// TIA Portal project "Esteira Properzi" (V15)

(* hardware
DEVICE "S7-1200 station_1"  S7-1200 Station
   slot 0: "Rack_0"  S7-1200 Rack  Rack  V1.0
   slot 1: "PLC_1"  CPU 1214C DC/DC/DC  6ES7 214-1AG40-0XB0  V4.2
*)

// ===== PLC "PLC_1"  CPU 1214C DC/DC/DC =====

VAR_GLOBAL   // PLC tag table "Default tag table"
   "Sensor Inicio Esteira" AT %I0.0 : Bool;
   "Sensor Meio Esteira" AT %I0.1 : Bool;
   "Sensor Fim Esteira" AT %I0.2 : Bool;
   "Sensor Nivel Alto Fusao" AT %I0.3 : Bool;
   "Sensor Nivel Medio Fusao" AT %I0.4 : Bool;
   "Sensor Nivel Baixo Fusao" AT %I0.5 : Bool;
   "Emergencia" AT %I0.6 : Bool;
   "Aut \ Man" AT %I0.7 : Bool;
   "Liga" AT %I1.0 : Bool;
   "Desliga" AT %I1.1 : Bool;
   "Motor" AT %Q0.0 : Bool;
   "Sinaleiro Verde" AT %Q0.1 : Bool;
   "Sinaleiro Vermelho" AT %Q0.2 : Bool;
   "Sonorizador" AT %Q0.3 : Bool;
   "Aux Sensor Inicio Esteira" AT %M2.0 : Bool;
   "Aux Sensor Meio Esteira" AT %M2.1 : Bool;
   "Aux Sensor Fim Esteira" AT %M2.2 : Bool;
   "Aux Sensor Nivel Alto Fusao" AT %M2.3 : Bool;
   "Aux Sensor Nivel Medio Fusao" AT %M2.4 : Bool;
   "Aux Sensor Nivel Baixo Fusao" AT %M2.5 : Bool;
   "System_Byte" AT %MB3 : Byte;
   "FirstScan" AT %M1.0 : Bool;
   "DiagStatusUpdate" AT %M1.1 : Bool;
   "AlwaysTRUE" AT %M1.2 : Bool;
   "AlwaysFALSE" AT %M1.3 : Bool;
   "Clock_Byte" AT %MB0 : Byte;
   "Clock_10Hz" AT %M0.0 : Bool;
   "Clock_5Hz" AT %M0.1 : Bool;
   "Clock_2.5Hz" AT %M0.2 : Bool;
   "Clock_2Hz" AT %M0.3 : Bool;
   "Clock_1.25Hz" AT %M0.4 : Bool;
   "Clock_1Hz" AT %M0.5 : Bool;
   "Clock_0.625Hz" AT %M0.6 : Bool;
   "Clock_0.5Hz" AT %M0.7 : Bool;
   "Aux Motor" AT %M4.0 : Bool;
   "Aux Sinaleiro Verde" AT %M4.1 : Bool;
   "Aux Sinaleiro Vermelho" AT %M4.2 : Bool;
   "Aux Sonorizador" AT %M4.3 : Bool;
   "Aux Emergencia" AT %M2.6 : Bool;
   "Aux Aut \ Man" AT %M2.7 : Bool;
   "Aux Liga" AT %M3.0 : Bool;
   "Aux Desliga" AT %M3.1 : Bool;
   "Auto" AT %M5.0 : Bool;
   "Pulso" AT %M1.4 : Bool;
   "Passo" AT %MW6 : Int;
   "Pulso 1" AT %M1.5 : Bool;
   "Pulso 2" AT %M1.6 : Bool;
   "Bomba" AT %Q0.4 : Bool;
   "Aux Bomba" AT %M1.7 : Bool;
   "Sensor Nivel Alto Operacao" AT %Q0.5 : Bool;
   "Sensor Nivel Medio Operacao" AT %Q0.6 : Bool;
   "Sensor Nivel Baixo Operacao" AT %Q0.7 : Bool;
   "Temperatura Zona Lingote Acima" AT %Q1.0 : Bool;
   "Temperatura Zona Bomba Abaixo" AT %Q1.3 : Bool;
   "Temperatura Zona Lingote Abaixo" AT %Q1.1 : Bool;
   "Temperatura Zona Bomba Acima" AT %Q1.2 : Bool;
   "Etapa" AT %MW8 : Int;
   "Aut \ Man Bomba" AT %I1.2 : Bool;
END_VAR

DATA_BLOCK "Alarmes_DB"   // DB5
{ S7_Optimized_Access := 'TRUE' }
VERSION : 0.1
// stored: InstanceOfName Alarmes
"Alarmes"
BEGIN
END_DATA_BLOCK

// folder: System blocks/Program resources

DATA_BLOCK "IEC_Timer_0_DB"   // DB1
{ S7_Optimized_Access := 'TRUE' }
AUTHOR : Simatic
FAMILY : IEC
NAME : IEC_TMR
VERSION : 1.0
// stored: InstanceOfName IEC_TIMER
"IEC_TIMER"
BEGIN
END_DATA_BLOCK

DATA_BLOCK "IEC_Timer_0_DB_1"   // DB2
{ S7_Optimized_Access := 'TRUE' }
AUTHOR : Simatic
FAMILY : IEC
NAME : IEC_TMR
VERSION : 1.0
// stored: InstanceOfName IEC_TIMER
"IEC_TIMER"
BEGIN
END_DATA_BLOCK

DATA_BLOCK "IEC_Timer_0_DB_2"   // DB3
{ S7_Optimized_Access := 'TRUE' }
AUTHOR : Simatic
FAMILY : IEC
NAME : IEC_TMR
VERSION : 1.0
// stored: InstanceOfName IEC_TIMER
"IEC_TIMER"
BEGIN
END_DATA_BLOCK

DATA_BLOCK "IEC_Timer_0_DB_3"   // DB4
{ S7_Optimized_Access := 'TRUE' }
AUTHOR : Simatic
FAMILY : IEC
NAME : IEC_TMR
VERSION : 1.0
// stored: InstanceOfName IEC_TIMER
"IEC_TIMER"
BEGIN
END_DATA_BLOCK

DATA_BLOCK "IEC_Timer_0_DB_4"   // DB6
{ S7_Optimized_Access := 'TRUE' }
AUTHOR : Simatic
FAMILY : IEC
NAME : IEC_TMR
VERSION : 1.0
// stored: InstanceOfName IEC_TIMER
"IEC_TIMER"
BEGIN
END_DATA_BLOCK

// folder: (top level)

FUNCTION_BLOCK "Alarmes"   // FB1, LAD
{ S7_Optimized_Access := 'TRUE' }
VERSION : 0.1
   VAR
      Temporizador : Array[0..10] of IEC_TIMER;
      tempo : Array[0..10] of Time;
   END_VAR
   VAR RETAIN
      Alarme : Array[0..16] of Bool;
   END_VAR
   VAR_TEMP   // added for the SCL form of the ladder/FBD networks
      _w1 : Bool;
   END_VAR
   // tempo[0] := T#200ms;
   // tempo[1] := T#100ms;
   // tempo[5] := T#200ms;
BEGIN

REGION Network 1: Temperaturas Fora do Range
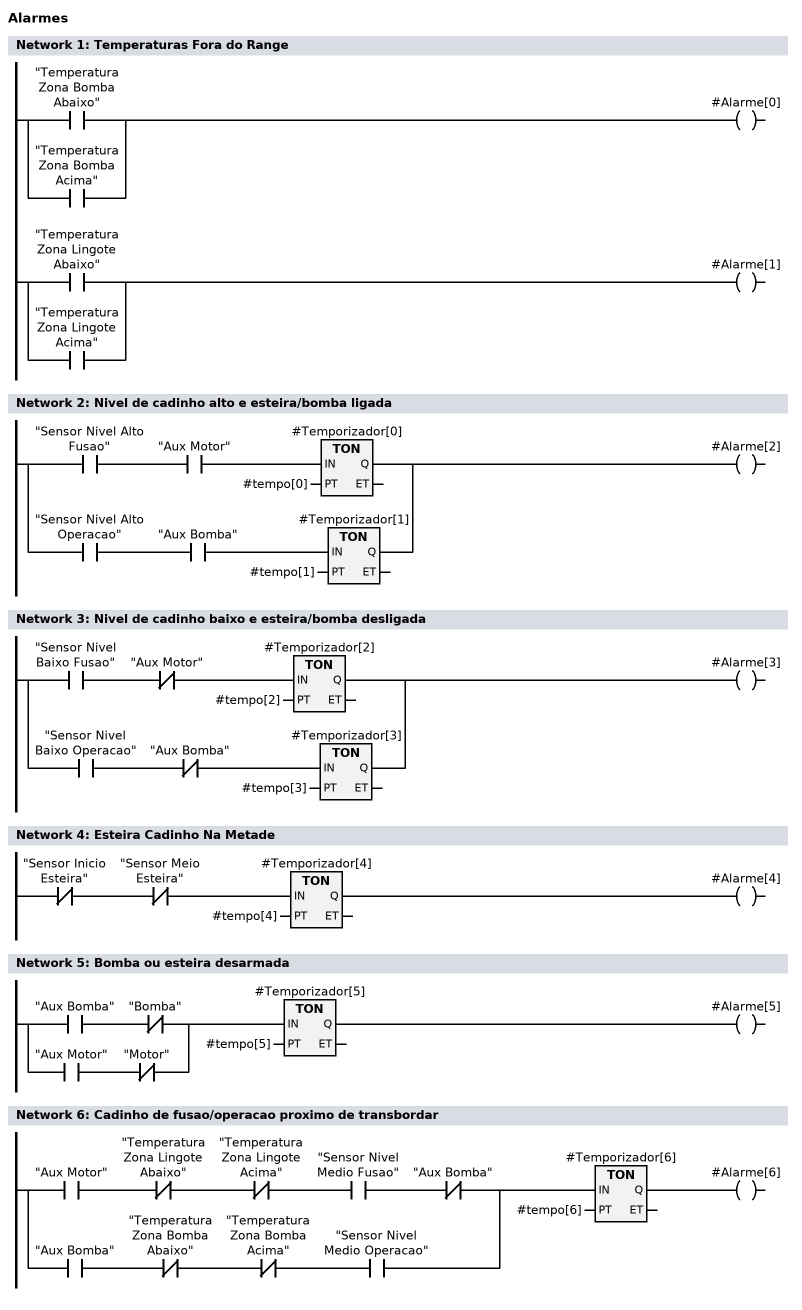
   RUNG wire#powerrail
      Contact( "Temperatura Zona Bomba Abaixo" )
      wire#w1
      Coil( #Alarme[0] )
   END_RUNG
   RUNG wire#powerrail
      Contact( "Temperatura Zona Bomba Acima" )
   END_RUNG wire#w1
   RUNG wire#powerrail
      Contact( "Temperatura Zona Lingote Abaixo" )
      wire#w2
      Coil( #Alarme[1] )
   END_RUNG
   RUNG wire#powerrail
      Contact( "Temperatura Zona Lingote Acima" )
   END_RUNG wire#w2
   // the same network as SCL:
   #Alarme[0] := "Temperatura Zona Bomba Abaixo" OR "Temperatura Zona Bomba Acima";
   #Alarme[1] := "Temperatura Zona Lingote Abaixo" OR "Temperatura Zona Lingote Acima";
END_REGION

REGION Network 2: Nivel de cadinho alto e esteira/bomba ligada
   #Temporizador[0].TON(IN := "Sensor Nivel Alto Fusao" AND "Aux Motor", PT := #tempo[0]);
   #_w1 := #Temporizador[0].Q;
   #Temporizador[1].TON(IN := "Sensor Nivel Alto Operacao" AND "Aux Bomba", PT := #tempo[1]);
   #Alarme[2] := #_w1 OR #Temporizador[1].Q;
END_REGION

REGION Network 3: Nivel de cadinho baixo e esteira/bomba desligada
   #Temporizador[2].TON(IN := "Sensor Nivel Baixo Fusao" AND NOT "Aux Motor", PT := #tempo[2]);
   #_w1 := #Temporizador[2].Q;
   #Temporizador[3].TON(IN := "Sensor Nivel Baixo Operacao" AND NOT "Aux Bomba", PT := #tempo[3]);
   #Alarme[3] := #_w1 OR #Temporizador[3].Q;
END_REGION

REGION Network 4: Esteira Cadinho Na Metade
   #Temporizador[4].TON(IN := NOT "Sensor Inicio Esteira" AND NOT "Sensor Meio Esteira", PT := #tempo[4]);
   #Alarme[4] := #Temporizador[4].Q;
END_REGION

REGION Network 5: Bomba ou esteira desarmada
   #Temporizador[5].TON(IN := ("Aux Bomba" AND NOT "Bomba") OR ("Aux Motor" AND NOT "Motor"), PT := #tempo[5]);
   #Alarme[5] := #Temporizador[5].Q;
END_REGION

REGION Network 6: Cadinho de fusao/operacao proximo de transbordar
   #Temporizador[6].TON(IN := ("Aux Motor" AND NOT "Temperatura Zona Lingote Abaixo" AND NOT "Temperatura Zona Lingote Acima" AND "Sensor Nivel Medio Fusao" AND NOT "Aux Bomba") OR ("Aux Bomba" AND NOT "Temperatura Zona Bomba Abaixo" AND NOT "Temperatura Zona Bomba Acima" AND "Sensor Nivel Medio Operacao"),
                        PT := #tempo[6]);
   #Alarme[6] := #Temporizador[6].Q;
END_REGION
END_FUNCTION_BLOCK

FUNCTION "Espelhamento Entradas" : Void   // FC1, LAD
{ S7_Optimized_Access := 'TRUE' }
VERSION : 0.1
BEGIN

REGION Network 1
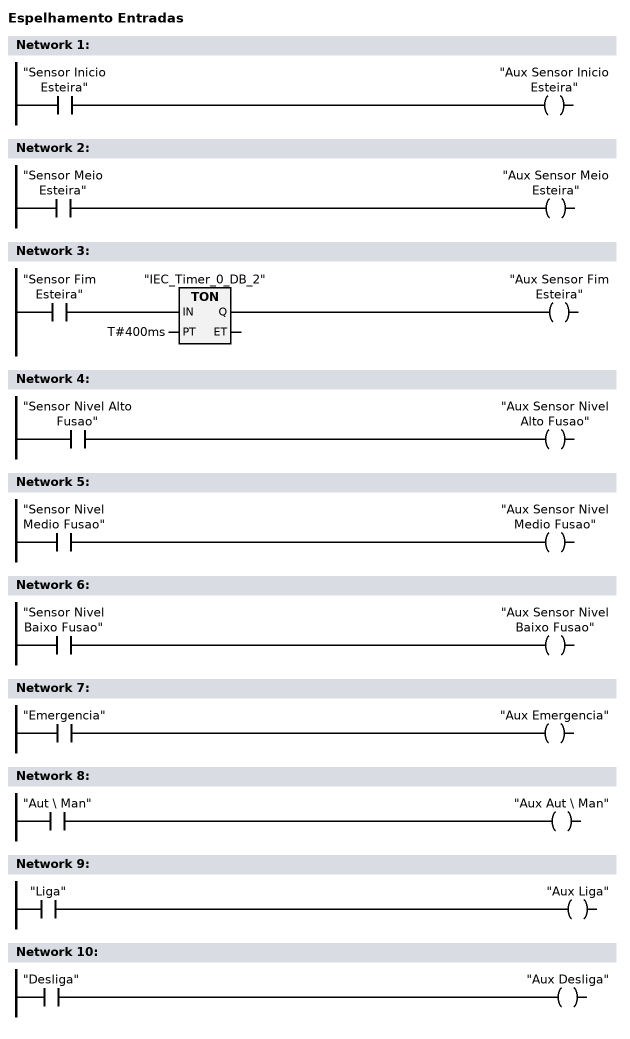
   RUNG wire#powerrail
      Contact( "Sensor Inicio Esteira" )
      Coil( "Aux Sensor Inicio Esteira" )
   END_RUNG
   // the same network as SCL:
   "Aux Sensor Inicio Esteira" := "Sensor Inicio Esteira";
END_REGION

REGION Network 2
   RUNG wire#powerrail
      Contact( "Sensor Meio Esteira" )
      Coil( "Aux Sensor Meio Esteira" )
   END_RUNG
   // the same network as SCL:
   "Aux Sensor Meio Esteira" := "Sensor Meio Esteira";
END_REGION

REGION Network 3
   "IEC_Timer_0_DB_2".TON(IN := "Sensor Fim Esteira", PT := T#400ms);
   "Aux Sensor Fim Esteira" := "IEC_Timer_0_DB_2".Q;
END_REGION

REGION Network 4
   RUNG wire#powerrail
      Contact( "Sensor Nivel Alto Fusao" )
      Coil( "Aux Sensor Nivel Alto Fusao" )
   END_RUNG
   // the same network as SCL:
   "Aux Sensor Nivel Alto Fusao" := "Sensor Nivel Alto Fusao";
END_REGION

REGION Network 5
   RUNG wire#powerrail
      Contact( "Sensor Nivel Medio Fusao" )
      Coil( "Aux Sensor Nivel Medio Fusao" )
   END_RUNG
   // the same network as SCL:
   "Aux Sensor Nivel Medio Fusao" := "Sensor Nivel Medio Fusao";
END_REGION

REGION Network 6
   RUNG wire#powerrail
      Contact( "Sensor Nivel Baixo Fusao" )
      Coil( "Aux Sensor Nivel Baixo Fusao" )
   END_RUNG
   // the same network as SCL:
   "Aux Sensor Nivel Baixo Fusao" := "Sensor Nivel Baixo Fusao";
END_REGION

REGION Network 7
   RUNG wire#powerrail
      Contact( "Emergencia" )
      Coil( "Aux Emergencia" )
   END_RUNG
   // the same network as SCL:
   "Aux Emergencia" := "Emergencia";
END_REGION

REGION Network 8
   RUNG wire#powerrail
      Contact( "Aut \ Man" )
      Coil( "Aux Aut \ Man" )
   END_RUNG
   // the same network as SCL:
   "Aux Aut \ Man" := "Aut \ Man";
END_REGION

REGION Network 9
   RUNG wire#powerrail
      Contact( "Liga" )
      Coil( "Aux Liga" )
   END_RUNG
   // the same network as SCL:
   "Aux Liga" := "Liga";
END_REGION

REGION Network 10
   RUNG wire#powerrail
      Contact( "Desliga" )
      Coil( "Aux Desliga" )
   END_RUNG
   // the same network as SCL:
   "Aux Desliga" := "Desliga";
END_REGION
END_FUNCTION

FUNCTION "Espelhamento Saida" : Void   // FC2, LAD
{ S7_Optimized_Access := 'TRUE' }
VERSION : 0.1
BEGIN

REGION Network 1
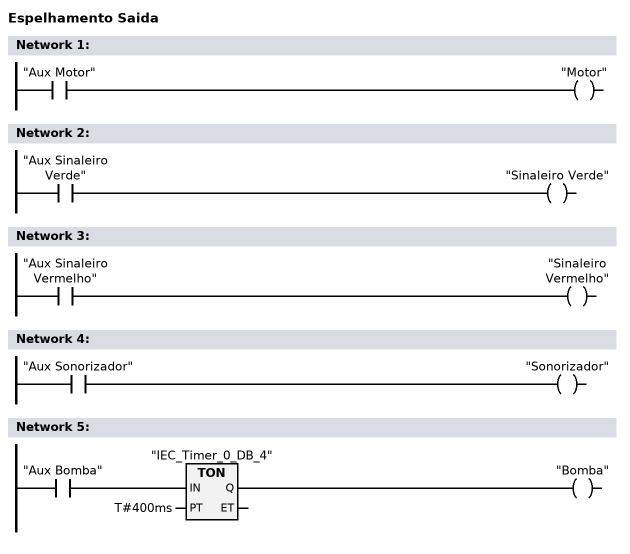
   RUNG wire#powerrail
      Contact( "Aux Motor" )
      Coil( "Motor" )
   END_RUNG
   // the same network as SCL:
   "Motor" := "Aux Motor";
END_REGION

REGION Network 2
   RUNG wire#powerrail
      Contact( "Aux Sinaleiro Verde" )
      Coil( "Sinaleiro Verde" )
   END_RUNG
   // the same network as SCL:
   "Sinaleiro Verde" := "Aux Sinaleiro Verde";
END_REGION

REGION Network 3
   RUNG wire#powerrail
      Contact( "Aux Sinaleiro Vermelho" )
      Coil( "Sinaleiro Vermelho" )
   END_RUNG
   // the same network as SCL:
   "Sinaleiro Vermelho" := "Aux Sinaleiro Vermelho";
END_REGION

REGION Network 4
   RUNG wire#powerrail
      Contact( "Aux Sonorizador" )
      Coil( "Sonorizador" )
   END_RUNG
   // the same network as SCL:
   "Sonorizador" := "Aux Sonorizador";
END_REGION

REGION Network 5
   "IEC_Timer_0_DB_4".TON(IN := "Aux Bomba", PT := T#400ms);
   "Bomba" := "IEC_Timer_0_DB_4".Q;
END_REGION
END_FUNCTION

FUNCTION "Manual" : Void   // FC3, LAD
{ S7_Optimized_Access := 'TRUE' }
VERSION : 0.1
BEGIN

REGION Network 1: Liga esteira cadinho de fusao
   // Botão liga ativado e cadinho de fusao não atingiu limite máximo
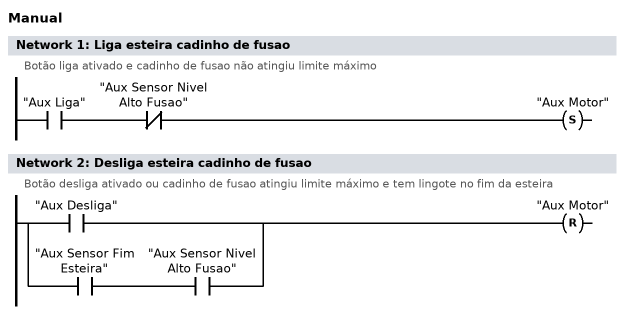
   RUNG wire#powerrail
      Contact( "Aux Liga" )
      I_Contact( "Aux Sensor Nivel Alto Fusao" )
      S_Coil( "Aux Motor" )
   END_RUNG
   // the same network as SCL:
   IF "Aux Liga" AND NOT "Aux Sensor Nivel Alto Fusao" THEN "Aux Motor" := TRUE; END_IF;
END_REGION

REGION Network 2: Desliga esteira cadinho de fusao
   // Botão desliga ativado ou cadinho de fusao atingiu limite máximo e tem lingote no fim da esteira
   RUNG wire#powerrail
      Contact( "Aux Desliga" )
      wire#w1
      R_Coil( "Aux Motor" )
   END_RUNG
   RUNG wire#powerrail
      Contact( "Aux Sensor Fim Esteira" )
      Contact( "Aux Sensor Nivel Alto Fusao" )
   END_RUNG wire#w1
   // the same network as SCL:
   IF "Aux Desliga" OR ("Aux Sensor Fim Esteira" AND "Aux Sensor Nivel Alto Fusao") THEN
       "Aux Motor" := FALSE;
   END_IF;
END_REGION
END_FUNCTION

FUNCTION "Automatico" : Void   // FC4, LAD
{ S7_Optimized_Access := 'TRUE' }
VERSION : 0.1
   VAR_TEMP   // added for the SCL form of the ladder/FBD networks
      _w1 : Bool;
   END_VAR
BEGIN

REGION Network 1: Botao Liga acionado -> Passo 1
   // Ativa sinaleiro verde
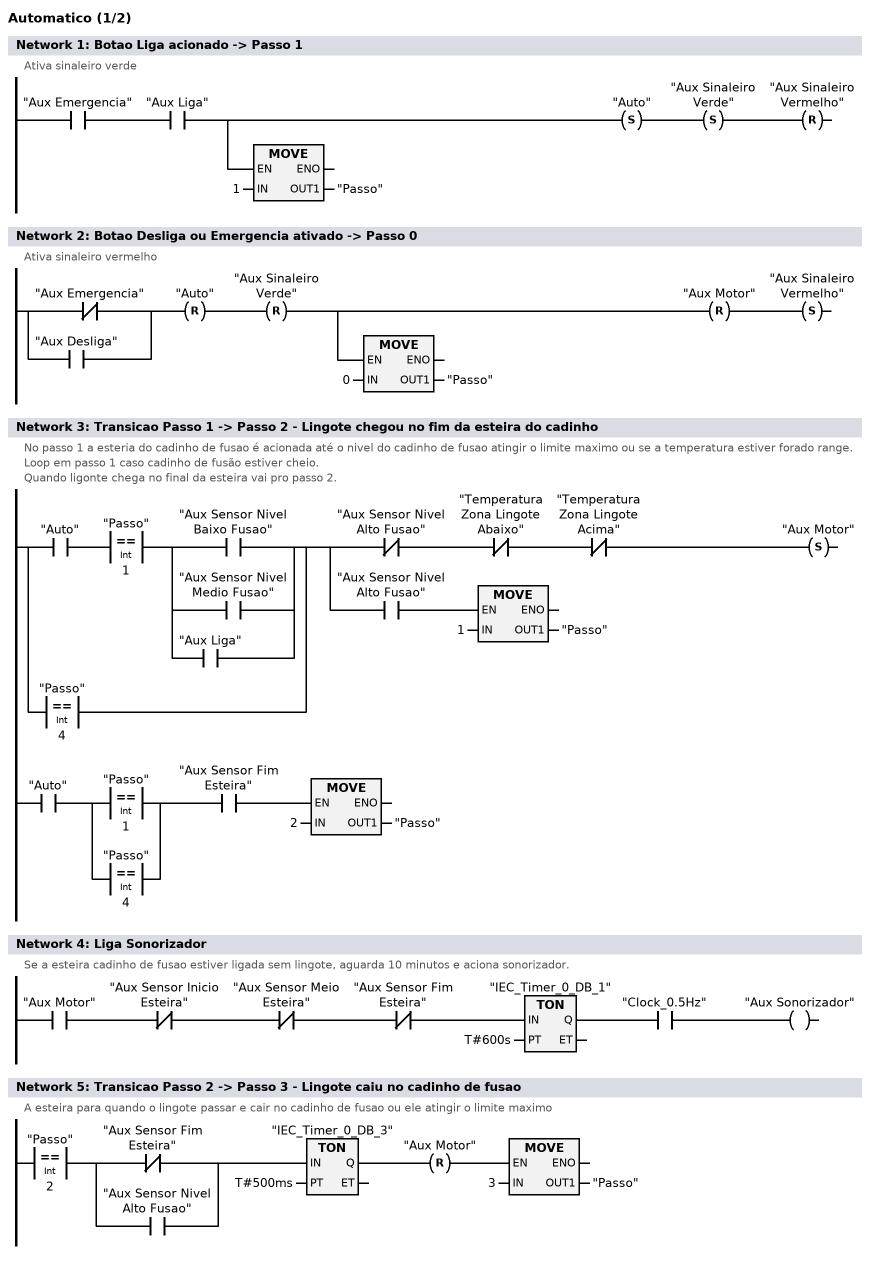
   RUNG wire#powerrail
      Contact( "Aux Emergencia" )
      Contact( "Aux Liga" )
      wire#w1
      S_Coil( "Auto" )
      S_Coil( "Aux Sinaleiro Verde" )
      R_Coil( "Aux Sinaleiro Vermelho" )
   END_RUNG
   RUNG wire#w1
      Move(in := 1, out1 => "Passo")
   END_RUNG
   // the same network as SCL:
   IF "Aux Emergencia" AND "Aux Liga" THEN
       "Auto" := TRUE;
       "Aux Sinaleiro Verde" := TRUE;
       "Aux Sinaleiro Vermelho" := FALSE;
       "Passo" := 1;
   END_IF;
END_REGION

REGION Network 2: Botao Desliga ou Emergencia ativado -> Passo 0
   // Ativa sinaleiro vermelho
   RUNG wire#powerrail
      I_Contact( "Aux Emergencia" )
      wire#w1
      R_Coil( "Auto" )
      R_Coil( "Aux Sinaleiro Verde" )
      wire#w2
      R_Coil( "Aux Motor" )
      S_Coil( "Aux Sinaleiro Vermelho" )
   END_RUNG
   RUNG wire#powerrail
      Contact( "Aux Desliga" )
   END_RUNG wire#w1
   RUNG wire#w2
      Move(in := 0, out1 => "Passo")
   END_RUNG
   // the same network as SCL:
   IF NOT "Aux Emergencia" OR "Aux Desliga" THEN
       "Auto" := FALSE;
       "Aux Sinaleiro Verde" := FALSE;
       "Aux Motor" := FALSE;
       "Aux Sinaleiro Vermelho" := TRUE;
       "Passo" := 0;
   END_IF;
END_REGION

REGION Network 3: Transicao Passo 1 -> Passo 2 - Lingote chegou no fim da esteira do cadinho
   // No passo 1 a esteria do cadinho de fusao é acionada até o nivel do cadinho de fusao atingir o limite maximo ou se a temperatura estiver forado range. Loop em passo 1 caso cadinho de fusão estiver cheio.
   // 
   // Quando ligonte chega no final da esteira vai pro passo 2.
   RUNG wire#powerrail
      Contact( "Auto" )
      { S7_Templates := "SrcType := Int" } EQ_Contact(in1 := "Passo", in2 := 1)
      wire#w1
      Contact( "Aux Sensor Nivel Baixo Fusao" )
      wire#w2
      I_Contact( "Aux Sensor Nivel Alto Fusao" )
      I_Contact( "Temperatura Zona Lingote Abaixo" )
      I_Contact( "Temperatura Zona Lingote Acima" )
      S_Coil( "Aux Motor" )
   END_RUNG
   RUNG wire#w1
      Contact( "Aux Sensor Nivel Medio Fusao" )
   END_RUNG wire#w2
   RUNG wire#w1
      Contact( "Aux Liga" )
   END_RUNG wire#w2
   RUNG wire#powerrail
      { S7_Templates := "SrcType := Int" } EQ_Contact(in1 := "Passo", in2 := 4)
   END_RUNG wire#w2
   RUNG wire#w2
      Contact( "Aux Sensor Nivel Alto Fusao" )
      Move(in := 1, out1 => "Passo")
   END_RUNG
   RUNG wire#powerrail
      Contact( "Auto" )
      wire#w3
      { S7_Templates := "SrcType := Int" } EQ_Contact(in1 := "Passo", in2 := 1)
      wire#w4
      Contact( "Aux Sensor Fim Esteira" )
      Move(in := 2, out1 => "Passo")
   END_RUNG
   RUNG wire#w3
      { S7_Templates := "SrcType := Int" } EQ_Contact(in1 := "Passo", in2 := 4)
   END_RUNG wire#w4
   // the same network as SCL:
   #_w1 := ("Auto" AND ("Passo" = 1) AND ("Aux Sensor Nivel Baixo Fusao" OR "Aux Sensor Nivel Medio Fusao" OR "Aux Liga")) OR ("Passo" = 4);
   IF #_w1 AND NOT "Aux Sensor Nivel Alto Fusao" AND NOT "Temperatura Zona Lingote Abaixo" AND NOT "Temperatura Zona Lingote Acima" THEN
       "Aux Motor" := TRUE;
   END_IF;
   IF #_w1 AND "Aux Sensor Nivel Alto Fusao" THEN "Passo" := 1; END_IF;
   IF "Auto" AND (("Passo" = 1) OR ("Passo" = 4)) AND "Aux Sensor Fim Esteira" THEN "Passo" := 2; END_IF;
END_REGION

REGION Network 4: Liga Sonorizador
   // Se a esteira cadinho de fusao estiver ligada sem lingote, aguarda 10 minutos e aciona sonorizador.
   "IEC_Timer_0_DB_1".TON(IN := "Aux Motor" AND NOT "Aux Sensor Inicio Esteira" AND NOT "Aux Sensor Meio Esteira" AND NOT "Aux Sensor Fim Esteira",
                          PT := T#600s);
   "Aux Sonorizador" := "IEC_Timer_0_DB_1".Q AND "Clock_0.5Hz";
END_REGION

REGION Network 5: Transicao Passo 2 -> Passo 3 - Lingote caiu no cadinho de fusao
   // A esteira para quando o lingote passar e cair no cadinho de fusao ou ele atingir o limite maximo
   "IEC_Timer_0_DB_3".TON(IN := ("Passo" = 2) AND (NOT "Aux Sensor Fim Esteira" OR "Aux Sensor Nivel Alto Fusao"),
                          PT := T#500ms);
   IF "IEC_Timer_0_DB_3".Q THEN
       "Aux Motor" := FALSE;
       "Passo" := 3;
   END_IF;
END_REGION

REGION Network 6: Transicao Passo 3 -> Passo 4 - Espera 20 segundos
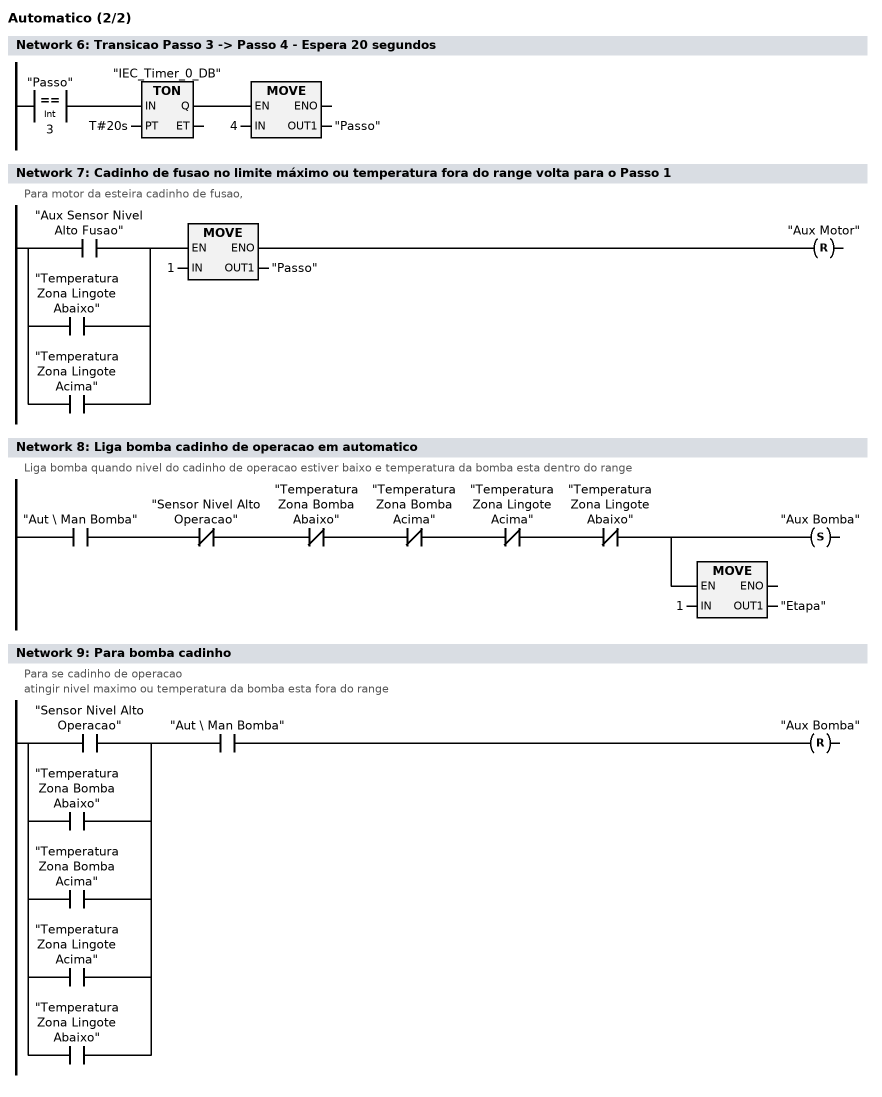
   "IEC_Timer_0_DB".TON(IN := "Passo" = 3, PT := T#20s);
   IF "IEC_Timer_0_DB".Q THEN "Passo" := 4; END_IF;
END_REGION

REGION Network 7: Cadinho de fusao no limite máximo ou temperatura fora do range volta para o Passo 1
   // Para motor da esteira cadinho de fusao,
   RUNG wire#powerrail
      Contact( "Aux Sensor Nivel Alto Fusao" )
      wire#w1
      Move(in := 1, out1 => "Passo")
      R_Coil( "Aux Motor" )
   END_RUNG
   RUNG wire#powerrail
      Contact( "Temperatura Zona Lingote Abaixo" )
   END_RUNG wire#w1
   RUNG wire#powerrail
      Contact( "Temperatura Zona Lingote Acima" )
   END_RUNG wire#w1
   // the same network as SCL:
   IF "Aux Sensor Nivel Alto Fusao" OR "Temperatura Zona Lingote Abaixo" OR "Temperatura Zona Lingote Acima" THEN
       "Passo" := 1;
       "Aux Motor" := FALSE;
   END_IF;
END_REGION

REGION Network 8: Liga bomba cadinho de operacao em automatico
   // Liga bomba quando nivel do cadinho de operacao estiver baixo e temperatura da bomba esta dentro do range
   RUNG wire#powerrail
      Contact( "Aut \ Man Bomba" )
      I_Contact( "Sensor Nivel Alto Operacao" )
      I_Contact( "Temperatura Zona Bomba Abaixo" )
      I_Contact( "Temperatura Zona Bomba Acima" )
      I_Contact( "Temperatura Zona Lingote Acima" )
      I_Contact( "Temperatura Zona Lingote Abaixo" )
      wire#w1
      S_Coil( "Aux Bomba" )
   END_RUNG
   RUNG wire#w1
      Move(in := 1, out1 => "Etapa")
   END_RUNG
   // the same network as SCL:
   IF "Aut \ Man Bomba" AND NOT "Sensor Nivel Alto Operacao" AND NOT "Temperatura Zona Bomba Abaixo" AND NOT "Temperatura Zona Bomba Acima" AND NOT "Temperatura Zona Lingote Acima" AND NOT "Temperatura Zona Lingote Abaixo" THEN
       "Aux Bomba" := TRUE;
       "Etapa" := 1;
   END_IF;
END_REGION

REGION Network 9: Para bomba cadinho
   // Para se cadinho de operacao 
   // atingir nivel maximo ou temperatura da bomba esta fora do range
   RUNG wire#powerrail
      Contact( "Sensor Nivel Alto Operacao" )
      wire#w1
      Contact( "Aut \ Man Bomba" )
      R_Coil( "Aux Bomba" )
   END_RUNG
   RUNG wire#powerrail
      Contact( "Temperatura Zona Bomba Abaixo" )
   END_RUNG wire#w1
   RUNG wire#powerrail
      Contact( "Temperatura Zona Bomba Acima" )
   END_RUNG wire#w1
   RUNG wire#powerrail
      Contact( "Temperatura Zona Lingote Acima" )
   END_RUNG wire#w1
   RUNG wire#powerrail
      Contact( "Temperatura Zona Lingote Abaixo" )
   END_RUNG wire#w1
   // the same network as SCL:
   IF ("Sensor Nivel Alto Operacao" OR "Temperatura Zona Bomba Abaixo" OR "Temperatura Zona Bomba Acima" OR "Temperatura Zona Lingote Acima" OR "Temperatura Zona Lingote Abaixo") AND "Aut \ Man Bomba" THEN
       "Aux Bomba" := FALSE;
   END_IF;
END_REGION
END_FUNCTION

ORGANIZATION_BLOCK "Main"   // OB1, LAD, ProgramCycle
TITLE = "Main Program Sweep (Cycle)"
{ S7_Optimized_Access := 'TRUE' }
VERSION : 0.1
   VAR_INPUT
      Initial_Call : Bool;   // Initial call of this OB
      Remanence : Bool;   // =True, if remanent data are available
   END_VAR
   VAR_TEMP   // added for the SCL form of the ladder/FBD networks
      _w1 : Bool;
      _w2 : Bool;
   END_VAR
BEGIN

REGION Network 1: Liga Automatico
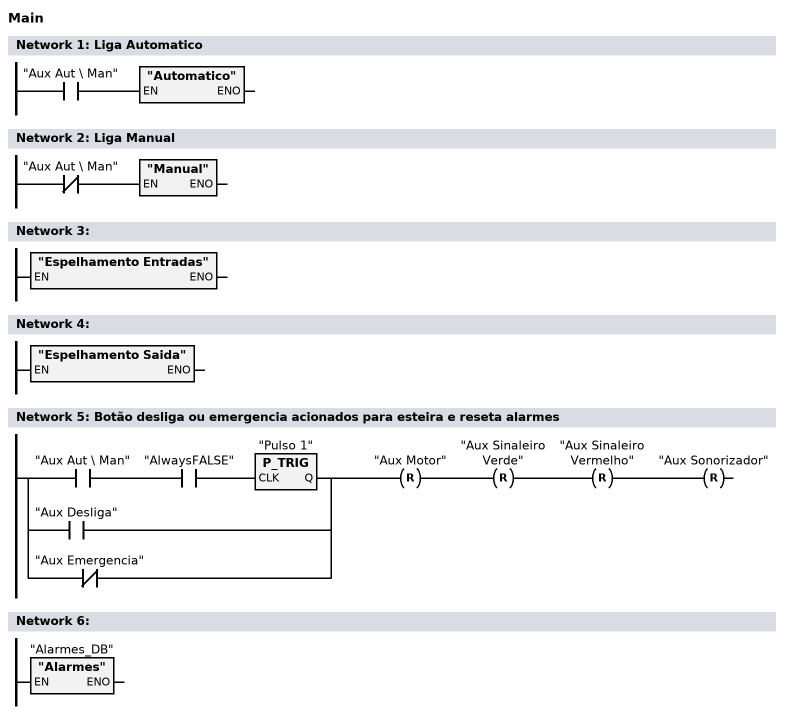
   RUNG wire#powerrail
      Contact( "Aux Aut \ Man" )
      "Automatico"()
   END_RUNG
   // the same network as SCL:
   IF "Aux Aut \ Man" THEN "Automatico"(); END_IF;
END_REGION

REGION Network 2: Liga Manual
   RUNG wire#powerrail
      I_Contact( "Aux Aut \ Man" )
      "Manual"()
   END_RUNG
   // the same network as SCL:
   IF NOT "Aux Aut \ Man" THEN "Manual"(); END_IF;
END_REGION

REGION Network 3
   RUNG wire#powerrail
      "Espelhamento Entradas"()
   END_RUNG
   // the same network as SCL:
   "Espelhamento Entradas"();
END_REGION

REGION Network 4
   RUNG wire#powerrail
      "Espelhamento Saida"()
   END_RUNG
   // the same network as SCL:
   "Espelhamento Saida"();
END_REGION

REGION Network 5: Botão desliga ou emergencia acionados para esteira e reseta alarmes
   RUNG wire#powerrail
      Contact( "Aux Aut \ Man" )
      Contact( "AlwaysFALSE" )
      P_Trig( "Pulso 1" )
      wire#w1
      R_Coil( "Aux Motor" )
      R_Coil( "Aux Sinaleiro Verde" )
      R_Coil( "Aux Sinaleiro Vermelho" )
      R_Coil( "Aux Sonorizador" )
   END_RUNG
   RUNG wire#powerrail
      Contact( "Aux Desliga" )
   END_RUNG wire#w1
   RUNG wire#powerrail
      I_Contact( "Aux Emergencia" )
   END_RUNG wire#w1
   // the same network as SCL:
   #_w1 := "Aux Aut \ Man" AND "AlwaysFALSE";
   #_w2 := #_w1 AND NOT "Pulso 1";   // rising edge
   "Pulso 1" := #_w1;
   IF #_w2 OR "Aux Desliga" OR NOT "Aux Emergencia" THEN
       "Aux Motor" := FALSE;
       "Aux Sinaleiro Verde" := FALSE;
       "Aux Sinaleiro Vermelho" := FALSE;
       "Aux Sonorizador" := FALSE;
   END_IF;
END_REGION

REGION Network 6
   RUNG wire#powerrail
      "Alarmes_DB"()
   END_RUNG
   // the same network as SCL:
   "Alarmes_DB"();   // "Alarmes"
END_REGION
END_ORGANIZATION_BLOCK